// TwinCAT 3 PLC project plc_lfe_motion_kmono
// ProgramVersion: 3.1.4022.7
// libraries:
//   Tc2_Standard, * (Beckhoff Automation GmbH)
//   Tc2_System, * (Beckhoff Automation GmbH)
//   Tc3_Module, * (Beckhoff Automation GmbH)
//   lcls-twincat-motion,0.0.0,SLAC
// project tree:
//   / PlcTask.TcTTO
//   POUs/ MAIN.TcPOU
// real-time tasks:
//   TASK PlcTask: cycle T#10ms, priority 20, ADS port 350
// motion (NC):
//   TASK NC-Task 1 SAF: cycle T#2ms, priority 4, ADS port 501
//   TASK NC-Task 1 SVB: cycle T#10ms, priority 8, ADS port 511
//   AXIS XTAL ANGLE X (id 1)
//     OtherSettings: AllowMotionCmdToSlave=true
//     encoder EncType=4
//       EncPara: MaxCount=#x0000ffff
//         Inc: RefSoftSyncMask=#x0000ffff
//     drive DrvType=24
//       Analog: ScaleFactorActTorque=0.1
//       TimeComp: TaskDelayCycles=1
//     controller CtrType=1
//       CtrPara: PriorControlFactor=1
//         PosDiffControl: Range=100
//         Observer: BandWidth=20
//   AXIS XTAL VERT Y (id 2)
//     Dynamic: DelayTime=0.008
//     Velo: SlowManual=3, FastManual=5, Maximum=5.08
//     OtherSettings: AllowMotionCmdToSlave=true, PulseDistancePos=0.5, PulseDistanceNeg=0.5
//     encoder EncType=7
//       EncPara: ScaleFactorNumerator=0.00172565918, MaxCount=#x0000ffff, ReferenceSystem=1
//         Inc: RefSoftSyncMask=#x0000ffff
//     drive DrvType=24
//       DrvPara: Inverse=true
//         Analog: VeloReferenz=50.8, ScaleFactorActTorque=0.1
//         TimeComp: TaskDelayCycles=1
//     controller CtrType=1
//       CtrPara: PriorControlFactor=1
//         PosDiffControl: Range=1
//         Observer: BandWidth=20
//   AXIS RETICLE HORIZ X (id 3)
//     Dynamic: DelayTime=0.008
//     Velo: RefSearch=3, RefSync=3, SlowManual=1, FastManual=3, Maximum=3
//     OtherSettings: AllowMotionCmdToSlave=true, PulseDistancePos=1, PulseDistanceNeg=1
//     encoder EncType=7
//       EncPara: ScaleFactorNumerator=0.0006942810059, MaxCount=#x0000ffff, ReferenceSystem=1
//         Inc: RefSoftSyncMask=#x0000ffff
//     drive DrvType=24
//       DrvPara: Inverse=true
//         Analog: VeloReferenz=6.35, ScaleFactorActTorque=0.1
//         TimeComp: TaskDelayCycles=1
//     controller CtrType=1
//       CtrPara: PriorControlFactor=1
//         PosDiffControl: Range=0.8
//         Observer: BandWidth=20
//   AXIS RETICLE VERT Y (id 4)
//     Dynamic: Acceleration=0.874139, Deceleration=0.178818, Jerk=152.824, DelayTime=0.008
//     Velo: RefSearch=2, RefSync=2, SlowManual=3, FastManual=5, Maximum=0.5
//     OtherSettings: AllowMotionCmdToSlave=true, PulseDistancePos=3, PulseDistanceNeg=3
//     encoder EncType=7
//       EncPara: ScaleFactorNumerator=0.004388516235, MaxCount=#x0000ffff, ReferenceSystem=1
//         Inc: RefSoftSyncMask=#x0000ffff
//     drive DrvType=24
//       Analog: VeloReferenz=10.16, ScaleFactorActTorque=0.1
//       TimeComp: TaskDelayCycles=1
//     controller CtrType=1
//       CtrPara: PriorControlFactor=1
//         PosDiffControl: Range=1.8
//         PID: PosKp=0
//         Observer: BandWidth=20
//   AXIS DIODE HORIZ X (id 5)
//     Dynamic: Acceleration=3.69082, Deceleration=3.69082, Jerk=68.11
//     Velo: SlowManual=1, FastManual=3, Maximum=4
//     OtherSettings: AllowMotionCmdToSlave=true, PulseDistancePos=1, PulseDistanceNeg=1
//     encoder EncType=7
//       EncPara: ScaleFactorNumerator=0.000711517334, MaxCount=#x0000ffff, ReferenceSystem=1
//         Inc: RefSoftSyncMask=#x0000ffff
//     drive DrvType=24
//       DrvPara: Inverse=true
//         Analog: VeloReferenz=6.35, ScaleFactorActTorque=0.1
//         TimeComp: TaskDelayCycles=1
//     controller CtrType=1
//       CtrPara: PriorControlFactor=1
//         PosDiffControl: Range=1
//         PID: PosKp=0.005
//         Observer: BandWidth=20
//   AXIS DIODE VERT Y (id 6)
//     Velo: SlowManual=2, FastManual=3, Maximum=4
//     OtherSettings: AllowMotionCmdToSlave=true
//     encoder EncType=7
//       EncPara: ScaleFactorNumerator=0.004388516235, MaxCount=#x0000ffff, ReferenceSystem=1
//         Inc: RefSoftSyncMask=#x0000ffff
//     drive DrvType=24
//       Analog: VeloReferenz=10.16, ScaleFactorActTorque=0.1
//       TimeComp: TaskDelayCycles=1
//     controller CtrType=1
//       CtrPara: PriorControlFactor=1
//         PosDiffControl: Range=1
//         Observer: BandWidth=20
// I/O:
//   DEVICE Device 2 (EtherCAT), AmsNetId 198.129.119.167.3.1
//     E0_MOTORS (EK1100) [EK1100 EtherCAT Coupler (2A E-Bus)]
//       E1_MOTORS (EL7031) [EL7031 1Ch. Stepper motor output stage (24V, 1.5A)]
//       E2_MOTORS (EL7041) [EL7041 1Ch. Stepper motor output stage (50V, 5A)]
//       E3_MOTORS (EL7041) [EL7041 1Ch. Stepper motor output stage (50V, 5A)]
//       E4_MOTORS (EL7041) [EL7041 1Ch. Stepper motor output stage (50V, 5A)]
//       E5_MOTORS (EL7041) [EL7041 1Ch. Stepper motor output stage (50V, 5A)]
//       E6_MOTORS (EL7041) [EL7041 1Ch. Stepper motor output stage (50V, 5A)]
//       ENDCAP_MOTORS (EL9011) [EL9011 End Terminal]
//     E0_LVDT (EK1100) [EK1100 EtherCAT Coupler (2A E-Bus)]
//       E1_LVDT(EL6021) [EL6021 Interface (RS422/485)]
//       E2_LVDT (EL1004)
//       E3_LVDT (EL1004)
//       E4_LVDT (EL3052) [EL3052 2Ch. Ana. Input 4-20mA]
//       E5_LVDT (EL3052) [EL3052 2Ch. Ana. Input 4-20mA]
//       E6_LVDT (EL3052)
//       ENDCAP_LVDT (EL9011) [EL9011 End Terminal]
// variable links:
//   (this object) <-> Device 2 (EtherCAT)/E0_MOTORS (EK1100)/E1_MOTORS (EL7031)
//     Drive/Inputs/In/nState1 @bit 3 <-> STM Status/Status/Error
//     Drive/Inputs/In/nState1 @bit 5 <-> STM Status/Status/Moving negative
//     Drive/Inputs/In/nState1 @bit 4 <-> STM Status/Status/Moving positive
//     Drive/Inputs/In/nState1 @bit 1 <-> STM Status/Status/Ready
//     Drive/Inputs/In/nState1 <-> STM Status/Status/Ready to enable
//     Drive/Inputs/In/nState1 @bit 6 <-> STM Status/Status/Torque reduced
//     Drive/Inputs/In/nState1 @bit 2 <-> STM Status/Status/Warning
//     Drive/Inputs/In/nState2 @bit 5 <-> STM Status/Status/Sync error
//     Drive/Inputs/In/nState2 @bit 7 <-> STM Status/Status/TxPDO Toggle
//     Drive/Inputs/In/nState4 @bit 1 <-> WcState/InputToggle
//     Drive/Inputs/In/nState4 <-> WcState/WcState
//     Drive/Outputs/Out/nCtrl1 <-> STM Control/Control/Enable
//     Drive/Outputs/Out/nCtrl1 @bit 2 <-> STM Control/Control/Reduce torque
//     Drive/Outputs/Out/nCtrl1 @bit 1 <-> STM Control/Control/Reset
//     Drive/Outputs/Out/nDataOut2[0] <-> STM Velocity/Velocity
//     Enc/Inputs/In/nDataIn1[0] <-> ENC Status compact/Counter value
//     Enc/Inputs/In/nDataIn2[0] <-> ENC Status compact/Latch value
//     Enc/Inputs/In/nState1 @bit 4 <-> ENC Status compact/Status/Counter overflow
//     Enc/Inputs/In/nState1 @bit 3 <-> ENC Status compact/Status/Counter underflow
//     Enc/Inputs/In/nState1 @bit 1 <-> ENC Status compact/Status/Latch extern valid
//     Enc/Inputs/In/nState1 @bit 2 <-> ENC Status compact/Status/Set counter done
//     Enc/Inputs/In/nState2 @bit 4 <-> ENC Status compact/Status/Status of extern latch
//     Enc/Inputs/In/nState2 @bit 5 <-> ENC Status compact/Status/Sync error
//     Enc/Inputs/In/nState2 @bit 7 <-> ENC Status compact/Status/TxPDO Toggle
//     Enc/Inputs/In/nState4 @bit 1 <-> WcState/InputToggle
//     Enc/Inputs/In/nState4 <-> WcState/WcState
//     Enc/Outputs/Out/nCtrl1 @bit 3 <-> ENC Control compact/Control/Enable latch extern on negative edge
//     Enc/Outputs/Out/nCtrl1 @bit 1 <-> ENC Control compact/Control/Enable latch extern on positive edge
//     Enc/Outputs/Out/nCtrl1 @bit 2 <-> ENC Control compact/Control/Set counter
//     Enc/Outputs/Out/nDataOut1[0] <-> ENC Control compact/Set counter value
//   (this object) <-> Device 2 (EtherCAT)/E0_LVDT (EK1100)/E4_LVDT (EL3052)
//     Enc/Inputs/In/nDataIn1[0] <-> AI Standard Channel 1/Value
//     Enc/Inputs/In/nDataIn1[0] <-> AI Standard Channel 2/Value
//     Enc/Inputs/In/nState4 @bit 1 <-> WcState/InputToggle
//     Enc/Inputs/In/nState4 <-> WcState/WcState
//   (this object) <-> Device 2 (EtherCAT)/E0_MOTORS (EK1100)/E2_MOTORS (EL7041)
//     Drive/Inputs/In/nState1 @bit 3 <-> STM Status/Status/Error
//     Drive/Inputs/In/nState1 @bit 5 <-> STM Status/Status/Moving negative
//     Drive/Inputs/In/nState1 @bit 4 <-> STM Status/Status/Moving positive
//     Drive/Inputs/In/nState1 @bit 1 <-> STM Status/Status/Ready
//     Drive/Inputs/In/nState1 <-> STM Status/Status/Ready to enable
//     Drive/Inputs/In/nState1 @bit 6 <-> STM Status/Status/Torque reduced
//     Drive/Inputs/In/nState1 @bit 2 <-> STM Status/Status/Warning
//     Drive/Inputs/In/nState2 @bit 5 <-> STM Status/Status/Sync error
//     Drive/Inputs/In/nState2 @bit 7 <-> STM Status/Status/TxPDO Toggle
//     Drive/Inputs/In/nState4 @bit 1 <-> WcState/InputToggle
//     Drive/Inputs/In/nState4 <-> WcState/WcState
//     Drive/Outputs/Out/nCtrl1 <-> STM Control/Control/Enable
//     Drive/Outputs/Out/nCtrl1 @bit 2 <-> STM Control/Control/Reduce torque
//     Drive/Outputs/Out/nCtrl1 @bit 1 <-> STM Control/Control/Reset
//     Drive/Outputs/Out/nDataOut2[0] <-> STM Velocity/Velocity
//   (this object) <-> Device 2 (EtherCAT)/E0_MOTORS (EK1100)/E3_MOTORS (EL7041)
//     Drive/Inputs/In/nState1 @bit 3 <-> STM Status/Status/Error
//     Drive/Inputs/In/nState1 @bit 5 <-> STM Status/Status/Moving negative
//     Drive/Inputs/In/nState1 @bit 4 <-> STM Status/Status/Moving positive
//     Drive/Inputs/In/nState1 @bit 1 <-> STM Status/Status/Ready
//     Drive/Inputs/In/nState1 <-> STM Status/Status/Ready to enable
//     Drive/Inputs/In/nState1 @bit 6 <-> STM Status/Status/Torque reduced
//     Drive/Inputs/In/nState1 @bit 2 <-> STM Status/Status/Warning
//     Drive/Inputs/In/nState2 @bit 5 <-> STM Status/Status/Sync error
//     Drive/Inputs/In/nState2 @bit 7 <-> STM Status/Status/TxPDO Toggle
//     Drive/Inputs/In/nState4 @bit 1 <-> WcState/InputToggle
//     Drive/Inputs/In/nState4 <-> WcState/WcState
//     Drive/Outputs/Out/nCtrl1 <-> STM Control/Control/Enable
//     Drive/Outputs/Out/nCtrl1 @bit 2 <-> STM Control/Control/Reduce torque
//     Drive/Outputs/Out/nCtrl1 @bit 1 <-> STM Control/Control/Reset
//     Drive/Outputs/Out/nDataOut2[0] <-> STM Velocity/Velocity
//   (this object) <-> Device 2 (EtherCAT)/E0_LVDT (EK1100)/E5_LVDT (EL3052)
//     Enc/Inputs/In/nDataIn1[0] <-> AI Standard Channel 1/Value
//     Enc/Inputs/In/nDataIn1[0] <-> AI Standard Channel 2/Value
//     Enc/Inputs/In/nState4 @bit 1 <-> WcState/InputToggle
//     Enc/Inputs/In/nState4 <-> WcState/WcState
//   (this object) <-> Device 2 (EtherCAT)/E0_MOTORS (EK1100)/E4_MOTORS (EL7041)
//     Drive/Inputs/In/nState1 @bit 3 <-> STM Status/Status/Error
//     Drive/Inputs/In/nState1 @bit 5 <-> STM Status/Status/Moving negative
//     Drive/Inputs/In/nState1 @bit 4 <-> STM Status/Status/Moving positive
//     Drive/Inputs/In/nState1 @bit 1 <-> STM Status/Status/Ready
//     Drive/Inputs/In/nState1 <-> STM Status/Status/Ready to enable
//     Drive/Inputs/In/nState1 @bit 6 <-> STM Status/Status/Torque reduced
//     Drive/Inputs/In/nState1 @bit 2 <-> STM Status/Status/Warning
//     Drive/Inputs/In/nState2 @bit 5 <-> STM Status/Status/Sync error
//     Drive/Inputs/In/nState2 @bit 7 <-> STM Status/Status/TxPDO Toggle
//     Drive/Inputs/In/nState4 @bit 1 <-> WcState/InputToggle
//     Drive/Inputs/In/nState4 <-> WcState/WcState
//     Drive/Outputs/Out/nCtrl1 <-> STM Control/Control/Enable
//     Drive/Outputs/Out/nCtrl1 @bit 2 <-> STM Control/Control/Reduce torque
//     Drive/Outputs/Out/nCtrl1 @bit 1 <-> STM Control/Control/Reset
//     Drive/Outputs/Out/nDataOut2[0] <-> STM Velocity/Velocity
//   (this object) <-> Device 2 (EtherCAT)/E0_MOTORS (EK1100)/E5_MOTORS (EL7041)
//     Drive/Inputs/In/nState1 @bit 3 <-> STM Status/Status/Error
//     Drive/Inputs/In/nState1 @bit 5 <-> STM Status/Status/Moving negative
//     Drive/Inputs/In/nState1 @bit 4 <-> STM Status/Status/Moving positive
//     Drive/Inputs/In/nState1 @bit 1 <-> STM Status/Status/Ready
//     Drive/Inputs/In/nState1 <-> STM Status/Status/Ready to enable
//     Drive/Inputs/In/nState1 @bit 6 <-> STM Status/Status/Torque reduced
//     Drive/Inputs/In/nState1 @bit 2 <-> STM Status/Status/Warning
//     Drive/Inputs/In/nState2 @bit 5 <-> STM Status/Status/Sync error
//     Drive/Inputs/In/nState2 @bit 7 <-> STM Status/Status/TxPDO Toggle
//     Drive/Inputs/In/nState4 @bit 1 <-> WcState/InputToggle
//     Drive/Inputs/In/nState4 <-> WcState/WcState
//     Drive/Outputs/Out/nCtrl1 <-> STM Control/Control/Enable
//     Drive/Outputs/Out/nCtrl1 @bit 2 <-> STM Control/Control/Reduce torque
//     Drive/Outputs/Out/nCtrl1 @bit 1 <-> STM Control/Control/Reset
//     Drive/Outputs/Out/nDataOut2[0] <-> STM Velocity/Velocity
//   (this object) <-> Device 2 (EtherCAT)/E0_LVDT (EK1100)/E6_LVDT (EL3052)
//     Enc/Inputs/In/nDataIn1[0] <-> AI Standard Channel 1/Value
//     Enc/Inputs/In/nState4 @bit 1 <-> WcState/InputToggle
//     Enc/Inputs/In/nState4 <-> WcState/WcState
//   (this object) <-> Device 2 (EtherCAT)/E0_MOTORS (EK1100)/E6_MOTORS (EL7041)
//     Drive/Inputs/In/nState1 @bit 3 <-> STM Status/Status/Error
//     Drive/Inputs/In/nState1 @bit 5 <-> STM Status/Status/Moving negative
//     Drive/Inputs/In/nState1 @bit 4 <-> STM Status/Status/Moving positive
//     Drive/Inputs/In/nState1 @bit 1 <-> STM Status/Status/Ready
//     Drive/Inputs/In/nState1 <-> STM Status/Status/Ready to enable
//     Drive/Inputs/In/nState1 @bit 6 <-> STM Status/Status/Torque reduced
//     Drive/Inputs/In/nState1 @bit 2 <-> STM Status/Status/Warning
//     Drive/Inputs/In/nState2 @bit 5 <-> STM Status/Status/Sync error
//     Drive/Inputs/In/nState2 @bit 7 <-> STM Status/Status/TxPDO Toggle
//     Drive/Inputs/In/nState4 @bit 1 <-> WcState/InputToggle
//     Drive/Inputs/In/nState4 <-> WcState/WcState
//     Drive/Outputs/Out/nCtrl1 <-> STM Control/Control/Enable
//     Drive/Outputs/Out/nCtrl1 @bit 2 <-> STM Control/Control/Reduce torque
//     Drive/Outputs/Out/nCtrl1 @bit 1 <-> STM Control/Control/Reset
//     Drive/Outputs/Out/nDataOut2[0] <-> STM Velocity/Velocity
//   plc_lfe_motion_kmono Instance <-> Device 2 (EtherCAT)/E0_MOTORS (EK1100)/E1_MOTORS (EL7031)
//     PlcTask Inputs/MAIN.bM1CCWLimit <-> STM Status/Status/Digital input 2
//     PlcTask Inputs/MAIN.bM1CWLimit <-> STM Status/Status/Digital input 1
//   plc_lfe_motion_kmono Instance <-> Device 2 (EtherCAT)/E0_MOTORS (EK1100)/E2_MOTORS (EL7041)
//     PlcTask Inputs/MAIN.bM2CCWLimit <-> STM Status/Status/Digital input 2
//     PlcTask Inputs/MAIN.bM2CWLimit <-> STM Status/Status/Digital input 1
//   plc_lfe_motion_kmono Instance <-> Device 2 (EtherCAT)/E0_MOTORS (EK1100)/E3_MOTORS (EL7041)
//     PlcTask Inputs/MAIN.bM3CCWLimit <-> STM Status/Status/Digital input 2
//     PlcTask Inputs/MAIN.bM3CWLimit <-> STM Status/Status/Digital input 1
//   plc_lfe_motion_kmono Instance <-> Device 2 (EtherCAT)/E0_MOTORS (EK1100)/E4_MOTORS (EL7041)
//     PlcTask Inputs/MAIN.bM4CCWLimit <-> STM Status/Status/Digital input 2
//     PlcTask Inputs/MAIN.bM4CWLimit <-> STM Status/Status/Digital input 1
//   plc_lfe_motion_kmono Instance <-> Device 2 (EtherCAT)/E0_MOTORS (EK1100)/E5_MOTORS (EL7041)
//     PlcTask Inputs/MAIN.bM5CCWLimit <-> STM Status/Status/Digital input 2
//     PlcTask Inputs/MAIN.bM5CWLimit <-> STM Status/Status/Digital input 1
//   plc_lfe_motion_kmono Instance <-> Device 2 (EtherCAT)/E0_MOTORS (EK1100)/E6_MOTORS (EL7041)
//     PlcTask Inputs/MAIN.bM6CCWLimit <-> STM Status/Status/Digital input 2
//     PlcTask Inputs/MAIN.bM6CWLimit <-> STM Status/Status/Digital input 1
//   plc_lfe_motion_kmono Instance <-> NC-Task 1 SAF/Axes/DIODE HORIZ X
//     PlcTask Inputs/MAIN.M5.Axis.NcToPlc <-> Outputs/ToPlc
//     PlcTask Outputs/MAIN.M5.Axis.PlcToNc <-> Inputs/FromPlc
//   plc_lfe_motion_kmono Instance <-> NC-Task 1 SAF/Axes/DIODE VERT Y
//     PlcTask Inputs/MAIN.M6.Axis.NcToPlc <-> Outputs/ToPlc
//     PlcTask Outputs/MAIN.M6.Axis.PlcToNc <-> Inputs/FromPlc
//   plc_lfe_motion_kmono Instance <-> NC-Task 1 SAF/Axes/RETICLE HORIZ X
//     PlcTask Inputs/MAIN.M3.Axis.NcToPlc <-> Outputs/ToPlc
//     PlcTask Outputs/MAIN.M3.Axis.PlcToNc <-> Inputs/FromPlc
//   plc_lfe_motion_kmono Instance <-> NC-Task 1 SAF/Axes/RETICLE VERT Y
//     PlcTask Inputs/MAIN.M4.Axis.NcToPlc <-> Outputs/ToPlc
//     PlcTask Outputs/MAIN.M4.Axis.PlcToNc <-> Inputs/FromPlc
//   plc_lfe_motion_kmono Instance <-> NC-Task 1 SAF/Axes/XTAL ANGLE X
//     PlcTask Inputs/MAIN.M1.Axis.NcToPlc <-> Outputs/ToPlc
//     PlcTask Outputs/MAIN.M1.Axis.PlcToNc <-> Inputs/FromPlc
//   plc_lfe_motion_kmono Instance <-> NC-Task 1 SAF/Axes/XTAL VERT Y
//     PlcTask Inputs/MAIN.M2.Axis.NcToPlc <-> Outputs/ToPlc
//     PlcTask Outputs/MAIN.M2.Axis.PlcToNc <-> Inputs/FromPlc

CONFIGURATION plc_lfe_motion_kmono
    RESOURCE PLC ON TwinCAT3
        TASK PlcTask(INTERVAL := T#10ms, PRIORITY := 20);
        PROGRAM MAIN WITH PlcTask : MAIN;
    END_RESOURCE
END_CONFIGURATION

// ---- POUs/MAIN.TcPOU
PROGRAM MAIN
VAR
	M1: DUT_MotionStage:=(nCommand:=3);
	M2: DUT_MotionStage:=(nCommand:=3);
	M3: DUT_MotionStage:=(nCommand:=3);
	M4: DUT_MotionStage:=(nCommand:=3);
	M5: DUT_MotionStage:=(nCommand:=3);
	M6: DUT_MotionStage:=(nCommand:=3);
	fbMotion1: FB_MotionStage;
	fbMotion2: FB_MotionStage;
	fbMotion3: FB_MotionStage;
	fbMotion4: FB_MotionStage;
	fbMotion5: FB_MotionStage;
	fbMotion6: FB_MotionStage;
	bM1CWLimit	AT 	%I*	:	BOOL;
	bM1CCWLimit	AT 	%I*	:	BOOL;
	bM2CWLimit	AT 	%I*	:	BOOL;
	bM2CCWLimit	AT 	%I*	:	BOOL;
	bM3CWLimit	AT 	%I*	:	BOOL;
	bM3CCWLimit	AT 	%I*	:	BOOL;
	bM4CWLimit	AT 	%I*	:	BOOL;
	bM4CCWLimit	AT 	%I*	:	BOOL;
	bM5CWLimit	AT 	%I*	:	BOOL;
	bM5CCWLimit	AT 	%I*	:	BOOL;
	bM6CWLimit	AT 	%I*	:	BOOL;
	bM6CCWLimit	AT 	%I*	:	BOOL;
	iM2Encoder 	AT	%I*	:	INT;
	iM3Encoder 	AT	%I*	:	INT;
	iM4Encoder 	AT	%I*	:	INT;
	iM5Encoder 	AT	%I*	:	INT;
	iM6Encoder 	AT	%I*	:	INT;
END_VAR

// Motor 1 XTAL ANGLE X (SP1L0-KMONO-MMS-01)
M1.bLimitForwardEnable 	:= bM1CWLimit;	//TRUE
M1.bLimitBackwardEnable := bM1CWLimit;	//TRUE
M1.nEnableMode 			:= Enum_StageEnableMode.STAGE_ENABLE_ALWAYS;
M1.bHardwareEnable		:= TRUE;
M1.bPowerSelf			:= TRUE;
fbMotion1(stMotionStage:=M1);

// Motor 2 XTAL VERT Y (SP1L0-KMONO-MMS-02)
M2.bLimitForwardEnable 	:= bM2CCWLimit;	//(+Y)
M2.bLimitBackwardEnable := bM2CWLimit;	//(-Y)
M2.nEnableMode 			:= Enum_StageEnableMode.STAGE_ENABLE_ALWAYS;
M2.bHardwareEnable		:= TRUE;
M2.bPowerSelf			:= TRUE;
fbMotion2(stMotionStage:=M2);

// Motor 3 RETICLE HORIZ X (SP1L0-KMONO-MMS-03)
M3.bLimitForwardEnable 	:= bM3CCWLimit;	//(+X)
M3.bLimitBackwardEnable := bM3CWLimit;	//(-X)
M3.nEnableMode 			:= Enum_StageEnableMode.STAGE_ENABLE_ALWAYS;
M3.bHardwareEnable		:= TRUE;
M3.bPowerSelf			:= TRUE;
fbMotion3(stMotionStage:=M3);

// Motor 4 RETICLE VERT Y (SP1L0-KMONO-MMS-04)
M4.bLimitForwardEnable 	:= bM4CWLimit;	//(+Y)
M4.bLimitBackwardEnable := bM4CCWLimit;	//(-Y)
M4.nEnableMode 			:= Enum_StageEnableMode.STAGE_ENABLE_ALWAYS;
M4.bHardwareEnable		:= TRUE;
M4.bPowerSelf			:= TRUE;
fbMotion4(stMotionStage:=M4);

// Motor 5 DIODE HORIZ X (SP1L0-KMONO-MMS-05)
M5.bLimitForwardEnable 	:= bM5CCWLimit;	//(+X)
M5.bLimitBackwardEnable := bM5CWLimit;	//(-X)
M5.nEnableMode 			:= Enum_StageEnableMode.STAGE_ENABLE_ALWAYS;
M5.bHardwareEnable		:= TRUE;
M5.bPowerSelf			:= TRUE;
fbMotion5(stMotionStage:=M5);

// Motor 6 DIODE VERT Y (SP1L0-KMONO-MMS-06)
M6.bLimitForwardEnable 	:= bM6CWLimit;	//(+Y)
M6.bLimitBackwardEnable := bM6CCWLimit;	//(-Y)
M6.nEnableMode 			:= Enum_StageEnableMode.STAGE_ENABLE_ALWAYS;
M6.bHardwareEnable		:= TRUE;
M6.bPowerSelf			:= TRUE;
fbMotion6(stMotionStage:=M6);

END_PROGRAM
